PROGRAM MAIN
VAR
	XboxController				: FB_Xbox_Controller('',1);
	
	XPlanarMover				: FB_XPlanarMoverStandard;
	bEnableMover				: BOOL := TRUE;

	
	fbXbox_2D_Joystick_XPlanar	: FB_Xbox_2D_Joystick_XPlanar;
	stOptions					: ST_Xbox_2D_Joystick_XPlanar_Options;
	bEnableJog					: BOOL;
	eJogMode					: E_Xbox_XPlanar_JogMode;
END_VAR

XPlanarMover.Cycle();
XboxController.Cycle();

IF bEnableMover THEN
	XPlanarMover.Enable(slogMessage := 'Enabling Mover');
	IF XPlanarMover.P_Enable.Done THEN
		bEnableMover := FALSE;
	END_IF
END_IF


stOptions.eJog_Mode 		:= eJogMode;
stOptions.fFastJog_Trigger 	:= XboxController.P_Left_Trigger;
stOptions.bFastJog_Button	:= XboxController.P_Buttons.bA_Button;

fbXbox_2D_Joystick_XPlanar.Jog(
								bEnable:= bEnableJog AND XboxController.P_Status.bConnected, 
								stJoystick:= XboxController.P_Left_Joystick, 
								xpMover:= XPlanarMover, 
								stOptions:= stOptions);

END_PROGRAM

(* stored: Version 1.1.0.1, ProductVersion 3.1.4024.11
   POU MAIN: Id {6229c1e7-7648-4318-a777-35026c64ff5c}, SpecialFunc None *)
